// TIA Portal V19 export
FUNCTION "FC_POS_TO_WORK" : Void   // FC53, STL
TITLE = Arbeitsdaten einlesen
{ S7_Optimized_Access := 'FALSE' }
AUTHOR : MS
// Überträgt die Positionsdaten zur Bearbeitung in den Bearbeitungs-DB
// stored: AutoNumber false
   VAR_INPUT
      Akt_Pos : USInt;   // Position die geladen wird
   END_VAR
   VAR_OUTPUT
      not_load : Bool;   // Position nicht laden
   END_VAR
BEGIN

NETWORK
TITLE = Copy Data
// Lädt Daten der aktuellen Position in Feld [0]
      L     "DB_POS".POS[#Akt_Pos].Typ;
      L     B#16#FF;
      ==I;
      =     #not_load;
      BEC;

      CALL  MOVE
      ( IN  := "DB_POS".POS[#Akt_Pos],
        OUT := "DB_POS".POS[0]
      );

END_FUNCTION
